{attribute addProperty BoxType "EL5101-0011-0016"}
{attribute addProperty Id "ENC_StatusAT %I*ENC_Status_481CA30A1620ENC_NextSync1TimeAT %I*ENC_NextSync1Time_4F9D66926480ENC_TxPdo_1_Samples_Counter_valueAT %I*ENC_TxPdo_1_Samples_Counter_value_730838783240ENC_ControlAT %Q*ENC_Control_015EAC9E4860WcStateAT %I*WcState_98A4DF7520.250InfoDataAT %I*InfoData_0BDED7BF144180"}
{attribute addProperty CRC "117001807"}
{attribute addProperty SizeInBites "306"}
{attribute addProperty SizeInBytes "38.25"}
TYPE EL5101_28E40609 :
STRUCT
	{attribute addProperty Name "ENC_Status"}
	ENC_Status : ENC_Status_481CA30A;
	{attribute addProperty Name "ENC_NextSync1Time"}
	ENC_NextSync1Time : ENC_NextSync1Time_4F9D6692;
	{attribute addProperty Name "ENC_TxPdo_1_Samples_Counter_value"}
	ENC_TxPdo_1_Samples_Counter_value : ENC_TxPdo_1_Samples_Counter_value_73083878;
	{attribute addProperty Name "ENC_Control"}
	ENC_Control : ENC_Control_015EAC9E;
	{attribute addProperty Name "WcState"}
	WcState : WcState_98A4DF75;
	{attribute addProperty Name "InfoData"}
	InfoData : InfoData_0BDED7BF;
END_STRUCT
END_TYPE

(* stored: Version 1.2.0.0, ProductVersion 3.1.4024.9
   DUT EL5101_28E40609: Id {d13832b5-f88a-4635-8dfc-76c57139c993} *)
